(*
    This functionblock acts as a stream buffer for use with FB_XmlControl
*)
FUNCTION_BLOCK FB_StreamBuffer 
VAR
    _PointerToStringBuffer : POINTER TO BYTE;
    _BufferSize : UDINT;
    _Length : UDINT;
END_VAR

(*
    Appends a string to the buffer
*)
PROPERTY Append : T_MaxString
SET
VAR
    ByteIn : POINTER TO BYTE;
    ByteBuffer : POINTER TO BYTE;
END_VAR
ByteIn := ADR(Append); 
ByteBuffer := _PointerToStringBuffer + _Length; // set start address

WHILE ByteIn^ <> 0 AND (_Length < _BufferSize ) DO
    ByteBuffer^ := ByteIn^; //Copy the 1st byte
    _Length := _Length + 1; // set new buffer length
    ByteIn := ByteIn + 1; // calculate new start address 
    ByteBuffer := ByteBuffer + 1; // calculate new start address 
END_WHILE;

ByteBuffer := _PointerToStringBuffer + _Length; // String End
ByteBuffer^ := 0; // null terminated string
END_SET
END_PROPERTY

(*
    Read current Buffersize
*)
PROPERTY BufferSize : UDINT
GET
BufferSize := _BufferSize;
END_GET
END_PROPERTY

(*  
    Clears the buffer and sets the length to 0
*)
METHOD PUBLIC Clear
VAR
	Count : UDINT;
END_VAR
IF (_PointerToStringBuffer = 0) OR (_BufferSize = 0) THEN
    RETURN;
END_IF

FOR Count := 0 TO (_BufferSize - 1) DO
    _PointerToStringBuffer[Count] := 0;
END_FOR

_Length := 0;
END_METHOD

(*
    Copies a string from the character buffer
*)
METHOD PUBLIC Copy : T_MaxString
VAR_INPUT
    StartPos : UDINT;
    EndPos : UDINT;
END_VAR
VAR_OUTPUT
    CopyLen : UDINT;
    XmlError : E_XmlError;
END_VAR
VAR
    Loop : UDINT;
    PointerToByteToCopy : POINTER TO BYTE;
    PointerToBuffer : POINTER TO BYTE;
    CurPos : UDINT;
END_VAR
Loop := 0;
PointerToByteToCopy := ADR(Copy);
PointerToBuffer := _PointerToStringBuffer + StartPos - 1;

WHILE(Loop < SIZEOF(Copy)) AND (StartPos - 1 + Loop < _Length) AND (StartPos + Loop < EndPos) DO
    PointerToByteToCopy^ := PointerToBuffer^;
    Loop := Loop + 1;
    PointerToByteToCopy := ADR(Copy) + Loop;
    PointerToBuffer := _PointerToStringBuffer + StartPos + Loop -1;
END_WHILE;

IF Loop = SIZEOF(Copy) THEN
    XmlError := E_XmlError.ErrorStringLen;
ELSIF StartPos - 1 + Loop = _Length THEN
    XmlError := E_XmlError.ErrorMaxBufferLen;
ELSE
    XmlError := E_XmlError.OK;
END_IF;

PointerToByteToCopy^ := 0;
CopyLen :=  Loop;
END_METHOD

METHOD PUBLIC CutOff : T_MaxString
VAR_INPUT
    StartPos : UDINT;
END_VAR
VAR_OUTPUT
    CutLen : UDINT; 
    XmlError : E_XmlError;
END_VAR
VAR
    Loop : UDINT;
    PointerToByteToCut : POINTER TO BYTE;
    PointerToByteBuffer : POINTER TO BYTE;
END_VAR
Loop := 0;
PointerToByteToCut := ADR(CutOff);
PointerToByteBuffer := _PointerToStringBuffer + StartPos - 1;

WHILE PointerToByteBuffer^ <> 0 AND(Loop < SIZEOF(CutOff)) AND StartPos -1  + Loop < _Length DO
    PointerToByteToCut^ := PointerToByteBuffer^;
    Loop := Loop + 1;
    PointerToByteToCut := ADR(CutOff) + Loop;
    PointerToByteBuffer := _PointerToStringBuffer + StartPos - 1 + Loop;
END_WHILE;

IF PointerToByteBuffer^ = 0 THEN
    XmlError := E_XmlError.OK;
ELSIF Loop = SIZEOF(CutOff) THEN
    XmlError := E_XmlError.ErrorStringLen;
ELSIF StartPos - 1 + Loop = _Length THEN
    XmlError := E_XmlError.ErrorMaxBufferLen;
END_IF;

PointerToByteToCut^ := 0;
_Length := StartPos -1;

PointerToByteBuffer := _PointerToStringBuffer + StartPos - 1;
PointerToByteBuffer^ := 0;

CutLen := Loop;
END_METHOD

(* 
    Find a searchstring in the buffer and returns its position.
    It's possible to add a preffered startposition within buffer
*)
METHOD PUBLIC Find : UDINT
VAR_INPUT
    SearchString : STRING;
    StartPos : UDINT;
END_VAR
VAR
    Loop : UDINT;
    Search : UDINT;
    PointerToBuffer : POINTER TO BYTE;
    PointerToSearch : POINTER TO BYTE;
END_VAR
Loop := 0;
Search := 0;

PointerToBuffer := _PointerToStringBuffer + StartPos;
PointerToSearch := ADR(SearchString);

WHILE(PointerToSearch^ <> 0 ) AND Loop + StartPos < _Length DO
    IF PointerToBuffer^ <> PointerToSearch^ THEN
        Loop := Loop + 1;
        PointerToBuffer := _PointerToStringBuffer + StartPos + Loop;
        PointerToSearch := ADR(SearchString);
        Search := 0;
    ELSE
        Search := Search + 1;
        PointerToBuffer := _PointerToStringBuffer + StartPos + Loop + Search;
        PointerToSearch := ADR(SearchString ) + Search;
    END_IF;
END_WHILE;
Find := Loop + 1 + StartPos;
END_METHOD

METHOD PUBLIC FindBack : UDINT
VAR_INPUT
    SearchString : T_MaxString;
END_VAR
VAR
    Loop : UDINT;
    Search : UDINT;
    PointerToBuffer : POINTER TO BYTE;
    PointerToSearch : POINTER TO BYTE;
END_VAR
Loop := 0;
Search := 0;

PointerToBuffer := _PointerToStringBuffer + _Length;
PointerToSearch := ADR(SearchString);

WHILE(PointerToSearch^ <> 0) AND Loop < _Length DO
    IF PointerToBuffer^ <> PointerToSearch^ THEN
        Loop := Loop + 1;
        PointerToBuffer := _PointerToStringBuffer + _Length - Loop;
        PointerToSearch := ADR(SearchString);
        Search := 0;
    ELSE
        Search := Search + 1;
        PointerToBuffer := _PointerToStringBuffer + _Length - Loop + Search;
        PointerToSearch := ADR(SearchString ) + Search;
    END_IF;
END_WHILE;
FindBack := _Length - Loop + 1;
END_METHOD

(*
    Gets/Sets the current length (in bytes) of the streambuffer
*)
PROPERTY Length : UDINT
GET
Length := _Length;
END_GET
SET
_Length := Length;
END_SET
END_PROPERTY

METHOD PUBLIC SetBuffer : BOOL;
VAR_INPUT
    PointerToBufferAddress : POINTER TO BYTE; // Set buffer address (ADR ...)
    SizeOfBuffer : UDINT; // Set buffer size (SIZEOF ...)
END_VAR
IF (PointerToBufferAddress = 0) OR (SizeOfBuffer = 0) THEN
    SetBuffer := FALSE;
    RETURN;
END_IF;

_BufferSize := SizeOfBuffer;
_PointerToStringBuffer := PointerToBufferAddress;

SetBuffer := TRUE;
END_METHOD

END_FUNCTION_BLOCK

(* stored: Version 1.1.0.1
   POU FB_StreamBuffer: Id {7f893efb-b056-43d3-9cf8-4965b865d1ab}, SpecialFunc None
   Property Append: Id {d4d616f0-7dc0-4c82-9980-a86820a4e603}
   Set Set: Id {773bf1db-6b9a-4581-be33-e4745bbc41df}
   Property BufferSize: Id {d2500465-6b5c-4fb0-9294-23ec2bd05ebc}
   Get Get: Id {41dc436d-8e79-4934-92fd-8311aee18e1d}
   Method Clear: Id {7b62bdfe-ea69-48e5-9767-e008c0e45b4f}
   Method Copy: Id {fd1ed528-0ae6-4cdf-afa3-b493b38da967}
   Method CutOff: Id {341d1e3e-5391-492c-b254-9eeda8f77da4}
   Method Find: Id {0c590575-e4a3-4c0d-a120-5741ea1d66bb}
   Method FindBack: Id {a337c425-1f09-4c1d-bd2b-84a002e37811}
   Property Length: Id {15fcf071-8b31-4039-8bff-7191e342bda2}
   Get Get: Id {d9ee832e-be82-4ebc-bf0b-bb382927ac05}
   Set Set: Id {1f4b0111-693f-45a7-87e0-f7d622425361}
   Method SetBuffer: Id {bbd47c2a-5140-429c-a3f1-6edaac587279} *)
